// TIA Portal V21 export
VAR_GLOBAL   // PLC tag table "K_Pid_Filler"
END_VAR
VAR_GLOBAL CONSTANT   // user constants
   K_Pid_Filler_TemperaturaPreparazioneProd : Int := 0;
END_VAR
